FUNCTION_BLOCK ANY2ANY_1156448476 (* Any to any conversion *)
  (* Standard: 61499-2 *)
  (* Version 1.0, 29.10.2008, marumil, nxtControl GmbH, Initial Version *)
  PACKAGE Main;
  (* Compiler Cpp *)
  {SET_ATTRIBUTE(Runtime.FBType.ImplementingType, Runtime.Standard#DYNGEN_ANY2ANY)}
  {SET_ATTRIBUTE(Configuration.GenericFBType.InterfaceParams, Runtime.Standard#CNT:=1;IN${CNT$}:STRING;OUT${CNT$}:INT)}
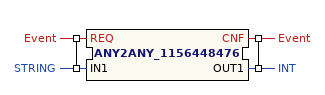
  EVENT_INPUT
    REQ WITH IN1; (* Normal Execution Request *)
  END_EVENT
  EVENT_OUTPUT
    CNF WITH OUT1; (* Execution Confirmation *)
  END_EVENT
  VAR_INPUT
    IN1 : STRING; (* Argument *)
  END_VAR
  VAR_OUTPUT
    OUT1 : INT; (* Result *)
  END_VAR
  EC_STATES
    START;
  END_STATES
END_FUNCTION_BLOCK
